TYPE DigitalOutputBase_1FE0D5EE :
STRUCT
END_STRUCT
END_TYPE

(* stored: Version 1.2.0.0, ProductVersion 3.1.4024.9
   DUT DigitalOutputBase_1FE0D5EE: Id {de6531af-7363-4e2b-8a3d-7843ee470a58} *)
